{attribute 'linkalways'} 
{attribute 'no_explicit_call' := 'This FB is a CLASS and must be accessed using methods or properties'}
{attribute 'enable_dynamic_creation'}
FUNCTION_BLOCK Node_F_VN_MinElementElementwise_TcVnVector2_UINT EXTENDS VisionNode
VAR
    ipContainer : _ITcVnContainer;
    aMin : _TcVnVector2_UINT;
    hrPrev : _HRESULT(S_OK);
    hresult : _HRESULT(S_OK);
END_VAR

METHOD PUBLIC  Clone : I_Node
VAR
	pNode : POINTER TO Node_F_VN_MinElementElementwise_TcVnVector2_UINT;
END_VAR
pNode := __NEW(Node_F_VN_MinElementElementwise_TcVnVector2_UINT);
Clone := pNode^;
END_METHOD

METHOD FB_init : BOOL
VAR_INPUT
	bInitRetains : BOOL; // if TRUE, the retain variables are initialized (warm start / cold start)
	bInCopyCode : BOOL;  // if TRUE, the instance afterwards gets moved into the copy code (online change)
END_VAR
AddInput('ipContainer', ipContainer);
AddInput('aMin', aMin);
AddInput('hrPrev', hrPrev);
AddOutput('ipContainer', ipContainer);
AddOutput('hresult',hresult);
END_METHOD

METHOD PROTECTED OnExecute : HRESULT
hresult.Value := F_VN_MinElementElementwise_TcVnVector2_UINT(
    ipContainer := ipContainer.Value,
    aMin := aMin.Value,
    hrPrev:= hrPrev.Value);
END_METHOD

METHOD PUBLIC PreExecutionCheck
VAR_INPUT
	Check : I_PreExecutionChecks;
END_VAR
Check.IsTrue(ipContainer.IsValid, 'ipContainer must be a valid container');
END_METHOD

END_FUNCTION_BLOCK

(* stored: Version 1.1.0.1, ProductVersion 3.1.4024.13
   POU Node_F_VN_MinElementElementwise_TcVnVector2_UINT: Id {45e283bd-6693-4d6f-a368-dd76be9b2727}, SpecialFunc None
   Folder Constructor: Id {8fad1abc-53f7-4215-ac31-e51a87abd89a}
   Method Clone: Id {4e751e26-f7fd-470f-a244-9508a8ace4d7}
   Method FB_init: Id {00b20f22-31c5-4ce2-8d8b-9985f0955dd9}
   Method OnExecute: Id {73a23d5e-ea71-4016-810a-ab148c44d60a}
   Method PreExecutionCheck: Id {a5903f73-9d9c-47b2-98c8-8b8f691aeaa3} *)
